TYPE STATE:
    STRUCT
        curTime: LREAL;
        cvar_c AT %Q*: LREAL;
        dvar_M_aut_r AT %Q*: LREAL;
        dvar_M_aut_b AT %Q*: BOOL;
        dvar_M_aut_i AT %Q*: DINT;
        dvar_M_aut_tii AT %Q*: TupleStruct_1;
        dvar_M_aut_i2 AT %Q*: DINT;
        dvar_M_aut_i3 AT %Q*: DINT;
        dvar_M_aut AT %Q*: enum_E;
    END_STRUCT
END_TYPE

(* stored: ProductVersion 3.1.0.18, Version 1.1.0.1 *)
